# EPICS substitutions: modules/event/evrSupport/Db/ioc/IOC-IN20-PM02evr.substitutions
#==============================================================================
#
# Abs:  LCLS EVR IOC records for IN20 PM02
#
# Name: IOC-IN20-PM02evr.substitutions
#
#==============================================================================
#
file evrPMXX.db
{
pattern { DEVICE        }
	{ EVR:IN20:PM02 }
}
